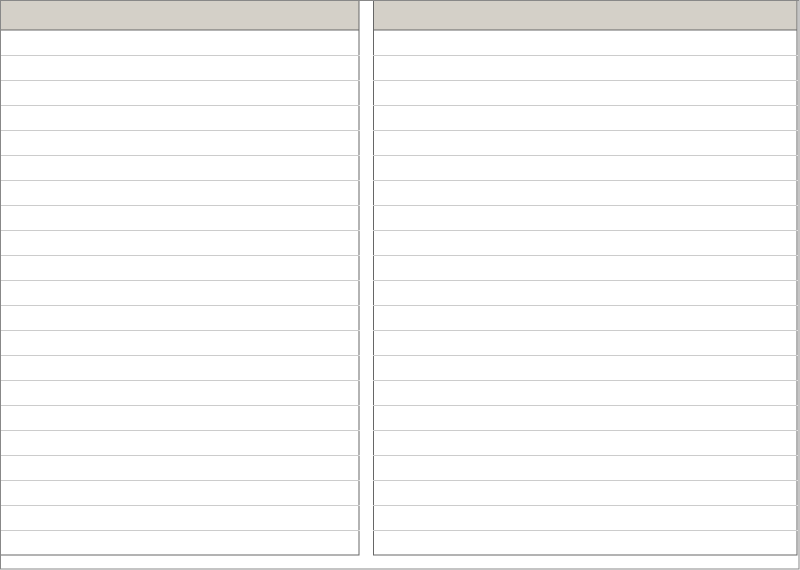
VISUALIZATION F99_IO_IO  // 800x570
    Table (0,0 359x555), data array: EL1809_M
        p1892666644: EL1809_M[2,INDEX]
        p338671338: EL1809_M[3,INDEX]
        p2685023577: EL1809_M[1,INDEX]
        Columns.Column.[0].Template: EL1809_M[1,INDEX]<>0
        Columns.Column.[1].Template: EL1809_M[2,INDEX]<>0
        Columns.Column.[2].Template: EL1809_M[3,INDEX]<>0
    Table (373,0 424x555), data array: EL2809_M
        p3854506369: EL2809_M[1,INDEX]
        p1892666644: EL2809_M[2,INDEX]
        p338671338: EL2809_M[3,INDEX]
        p2170511999: EL2809_M[4,INDEX]
        Columns.Column.[2].Template: EL2809_M[3,INDEX]<>0
        Columns.Column.[0].Template: EL2809_M[1,INDEX]<>0
        Columns.Column.[1].Template: EL2809_M[2,INDEX]<>0
        Columns.Column.[3].Template: EL2809_M[4,INDEX]<>0
END_VISUALIZATION

(* stored: Version 1.1.0.1, ProductVersion 3.1.4024.11
   Visu F99_IO_IO: Id {3cdbc7d0-05bf-42f9-9333-6abdf108d884} *)
